(* CODESYS project CintasSoplado.project
   Title: CintasSoplado
   Version: 0.0.0.0
   Author: serbogr1

Project tree, tasks and I/O mapping:
  MyController : TM241CE40R, Schneider Electric, order no. TM241CE40R, version 4.0.6.18
    application Application
      libraries: Toolbox, 2.2.0.0 (Schneider Electric); SysTime, 3.4.1.20 (System)
      task MAST (cyclic, interval 50 ms, priority 15) calls ProcesoUno, ProcesoDos, Pulsadores, PID, ControlSoplado, Gestion_HMI
      global variables GVL
      visualisation HMIW_Control
      image pool ImagePool
      program ProcesoDos [SFC]: E2_active, E10_active
      program PID [LD]
      program ProcesoUno [SFC]: E8_active, E7_active, E9_active, E10_active, E11_active, E12_active, E1_active
      program Pulsadores [LD]
      program ControlSoplado [SFC]: E1_active
      program Gestion_HMI [LD]
    DI : Digital Inputs, Schneider Electric, version 4.0.6.18
        input  idwDI_IDW0 : DWORD  // IDW0
        input  ibDI_IB1 : BYTE  // IB1
    DQ : Digital Outputs, Schneider Electric, version 4.0.6.18
        output qwDQ_QW0 : WORD  // QW0
        output qbDQ_QB1 : BYTE  // QB1
    Counters : Counters, Schneider Electric, version 4.0.6.18
    Pulse_Generators : Pulse Generators, Schneider Electric, version 4.0.6.18
    Cartridge_1 : Cartridge, Schneider Electric, version 4.0.6.18
      TMC4AI2 : TMC4AI2, Schneider Electric, order no. TMC4AI2, version 1.0.1.0
          input  iiTMC4AI2_IW0 : INT  // IW0
          input  iiTMC4AI2_IW1 : INT  // IW1
          input  ibTMC4AI2_IW2 : BYTE  // IW2
    Cartridge_2 : Cartridge, Schneider Electric, version 4.0.6.18
      TMC4AQ2 : TMC4AQ2, Schneider Electric, order no. TMC4AQ2, version 1.0.1.1
          output qiTMC4AQ2_QW0 : INT  // QW0
          output qiTMC4AQ2_QW1 : INT  // QW1
          input  ibTMC4AQ2_IW0 : BYTE  // IW0
    IO_Bus : IO bus - TM3, Schneider Electric, version 4.0.6.18
    COM_Bus : COM bus, Schneider Electric, version 4.0.6.18
    Ethernet_1 : Ethernet Network, Schneider Electric, version 4.0.6.18
        settings: WebServer = TRUE; FTP Server = TRUE; SoMachine Protocol = TRUE; Modbus Server = TRUE; NetManage Protocol = TRUE; SNMP protocol = TRUE; Enable Routing = FALSE; WebVisu protocol = TRUE; DHCP Server Active = FALSE
    Serial_Line_1 : Serial line, Schneider Electric, version 4.0.6.18
      SoMachine_Network_Manager : SoMachine-Network Manager, Schneider Electric, version 4.0.0.2
    Serial_Line_2 : Serial line, Schneider Electric, version 4.0.6.18
      Modbus_Manager : Modbus Manager, Schneider Electric, version 4.0.0.2
  text list GlobalTextList
*)

// MyController/Application/GVL
VAR_GLOBAL
END_VAR

// MyController/Application/ProcesoUno
PROGRAM ProcesoUno
VAR
	bS_FC_Empujador_1          AT %IX0.0: BOOL; (*I1*)
	bS_IC_Empujador_1          AT %IX0.1: BOOL; (*I2*)
	bS_FC_Empujador_2          AT %IX0.2: BOOL; (*I3*)
	bS_IC_Empujador_2          AT %IX0.3: BOOL; (*I4*)
	bS_FT_Empujador_1          AT %IX0.4: BOOL; (*I5*)
	bS_FT_Fresadora            AT %IX0.5: BOOL; (*I6*)
	bS_FT_Carga                AT %IX0.6: BOOL; (*I7*)
	bS_FT_Taladro              AT %IX0.7: BOOL; (*I8*)
	bS_FT_Salida               AT %IX1.0: BOOL; (*I9*)

	FalloSensores              AT %MX0.5: BOOL:=FALSE;;
	CintaFresadoraP1                    : BOOL;	
	CintaTaladroP1                      : BOOL;	
	CintaAlimentacionP1                 : BOOL;
	MotorFresadora                      : BOOL;
    bSiguientePieza            AT %MX0.4: BOOL; (*Activa cuando se puede poner la siguiente pieza*)
	iTiempoFresado                      : INT:=2;	
END_VAR

VAR_OUTPUT
	tEmpujador_1   : TIME:=T#1S;
	tFresado       : TIME:=T#1S;
END_VAR

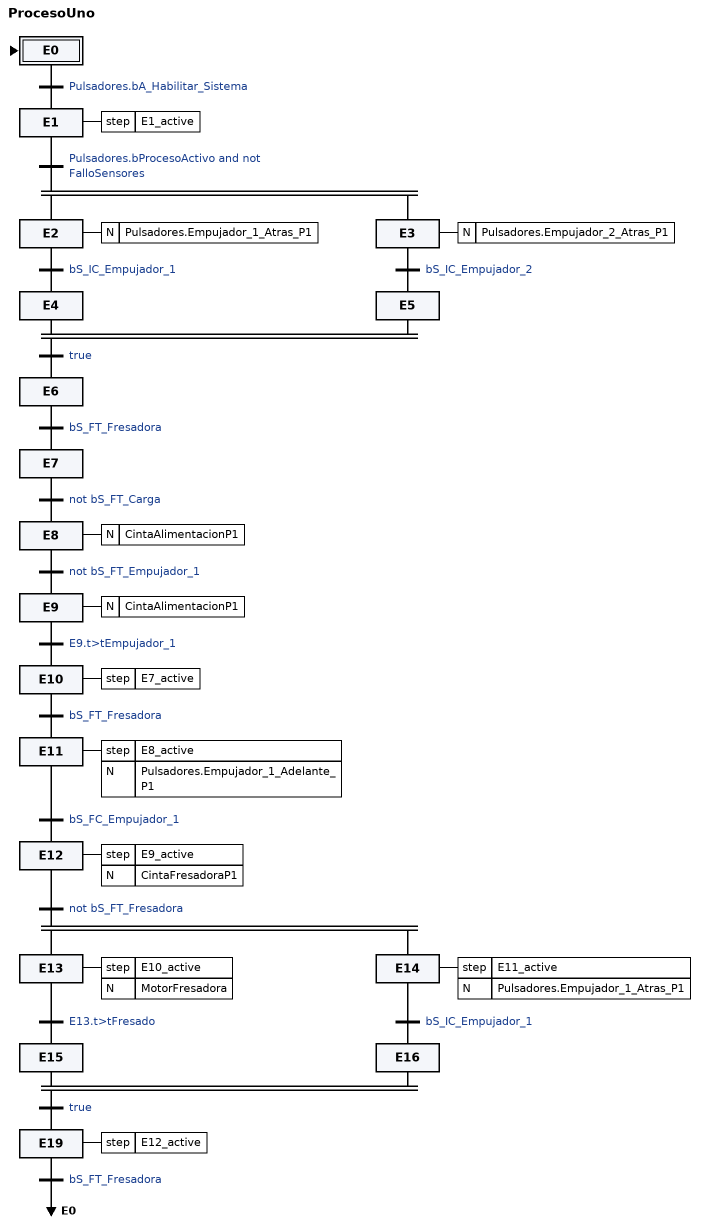
INITIAL_STEP E0:
END_STEP
TRANSITION FROM E0 TO E1
    := Pulsadores.bA_Habilitar_Sistema;
END_TRANSITION
STEP E1:
    E1_active(N);  // step action
END_STEP
TRANSITION FROM E1 TO (E2, E3)
    := Pulsadores.bProcesoActivo and not FalloSensores;
END_TRANSITION
STEP E2:
    Pulsadores.Empujador_1_Atras_P1(N);
END_STEP
TRANSITION FROM E2 TO E4
    := bS_IC_Empujador_1;
END_TRANSITION
STEP E4:
END_STEP
STEP E3:
    Pulsadores.Empujador_2_Atras_P1(N);
END_STEP
TRANSITION FROM E3 TO E5
    := bS_IC_Empujador_2;
END_TRANSITION
STEP E5:
END_STEP
TRANSITION FROM (E4, E5) TO E6
    := true;
END_TRANSITION
STEP E6:
END_STEP
TRANSITION FROM E6 TO E7
    := bS_FT_Fresadora;
END_TRANSITION
STEP E7:
END_STEP
TRANSITION FROM E7 TO E8
    := not bS_FT_Carga;
END_TRANSITION
STEP E8:
    CintaAlimentacionP1(N);
END_STEP
TRANSITION FROM E8 TO E9
    := not bS_FT_Empujador_1;
END_TRANSITION
STEP E9:
    CintaAlimentacionP1(N);
END_STEP
TRANSITION FROM E9 TO E10
    := E9.t>tEmpujador_1;
END_TRANSITION
STEP E10:
    E7_active(N);  // step action
END_STEP
TRANSITION FROM E10 TO E11
    := bS_FT_Fresadora;
END_TRANSITION
STEP E11:
    E8_active(N);  // step action
    Pulsadores.Empujador_1_Adelante_P1(N);
END_STEP
TRANSITION FROM E11 TO E12
    := bS_FC_Empujador_1;
END_TRANSITION
STEP E12:
    E9_active(N);  // step action
    CintaFresadoraP1(N);
END_STEP
TRANSITION FROM E12 TO (E13, E14)
    := not bS_FT_Fresadora;
END_TRANSITION
STEP E13:
    E10_active(N);  // step action
    MotorFresadora(N);
END_STEP
TRANSITION FROM E13 TO E15
    := E13.t>tFresado;
END_TRANSITION
STEP E15:
END_STEP
STEP E14:
    E11_active(N);  // step action
    Pulsadores.Empujador_1_Atras_P1(N);
END_STEP
TRANSITION FROM E14 TO E16
    := bS_IC_Empujador_1;
END_TRANSITION
STEP E16:
END_STEP
TRANSITION FROM (E15, E16) TO E19
    := true;
END_TRANSITION
STEP E19:
    E12_active(N);  // step action
END_STEP
TRANSITION FROM E19 TO E0
    := bS_FT_Fresadora;
END_TRANSITION

ACTION E8_active:
IF bS_FT_Carga THEN
	bSiguientePieza := TRUE;
ELSIF NOT bS_FT_Carga THEN
	bSiguientePieza := FALSE;
END_IF
END_ACTION

ACTION E7_active:
IF bS_FT_Carga THEN
	bSiguientePieza := TRUE;
ELSIF NOT bS_FT_Carga THEN
	bSiguientePieza := FALSE;
END_IF
END_ACTION

ACTION E9_active:
IF bS_FT_Carga THEN
	bSiguientePieza := TRUE;
ELSIF NOT bS_FT_Carga THEN
	bSiguientePieza := FALSE;
END_IF
END_ACTION

ACTION E10_active:
IF bS_FT_Carga THEN
	bSiguientePieza := TRUE;
ELSIF NOT bS_FT_Carga THEN
	bSiguientePieza := FALSE;
END_IF

IF Gestion_HMI.bSum_T_Fresado THEN
	iTiempoFresado := iTiempoFresado + 1;
END_IF
IF Gestion_HMI.bRes_T_Fresado THEN
	iTiempoFresado := iTiempoFresado - 1;
END_IF

	tFresado := INT_TO_TIME(iTiempoFresado*1000);
END_ACTION

ACTION E11_active:
IF bS_FT_Carga THEN
	bSiguientePieza := TRUE;
ELSIF NOT bS_FT_Carga THEN
	bSiguientePieza := FALSE;
END_IF
END_ACTION

ACTION E12_active:
IF bS_FT_Carga THEN
	bSiguientePieza := TRUE;
ELSIF NOT bS_FT_Carga THEN
	bSiguientePieza := FALSE;
END_IF
END_ACTION

ACTION E1_active:
IF NOT Pulsadores.bBotonInicioHMIW THEN
	IF NOT bS_FT_Carga THEN
		FalloSensores:=TRUE;	
	END_IF
	IF NOT bS_FT_Empujador_1 THEN
		FalloSensores:=TRUE;
	END_IF
	IF NOT bS_FT_Fresadora THEN
		FalloSensores:=TRUE;
	END_IF
	IF NOT bS_FT_Taladro THEN
		FalloSensores:=TRUE;
	END_IF
	IF NOT bS_FT_Salida THEN
		FalloSensores:=TRUE;	
	END_IF
	
	IF bS_FT_Carga AND bS_FT_Empujador_1 AND bS_FT_Fresadora AND bS_FT_Taladro AND bS_FT_Salida THEN
		FalloSensores:=FALSE;			
	END_IF
END_IF
END_ACTION

END_PROGRAM

// MyController/Application/Gestion_HMI
PROGRAM Gestion_HMI
VAR
	bSum_T_Fresado              AT %MX3.0: BOOL;
	bRes_T_Fresado              AT %MX3.1: BOOL;
	bSum_T_Taladrado            AT %MX3.2: BOOL;
	bRes_T_Taladrado            AT %MX3.3: BOOL;
	bSum_T_Soplado              AT %MX3.4: BOOL;
	bRes_T_Soplado              AT %MX3.5: BOOL;		
	bSum_AnguloInicio           AT %MX3.6: BOOL;		
	bRes_AnguloInicio           AT %MX3.7: BOOL;
	bSum_AnguloSoplado          AT %MX4.0: BOOL;
	bRes_AnguloSoplado          AT %MX4.1: BOOL;	

	bSe_FC_Empujador_1          AT %MX0.6: BOOL; (*Posición de pieza según el sensor en la HMI*)
	bSe_FC_Empujador_2          AT %MX0.7: BOOL; 
	bSe_FT_Empujador_1          AT %MX1.0: BOOL; 
	bSe_FT_Fresadora            AT %MX1.2: BOOL; 
	bSe_FT_Carga                AT %MX1.3: BOOL; 
	bSe_FT_Taladro              AT %MX1.4: BOOL; 
	bSe_FT_Salida               AT %MX1.5: BOOL; 
	
	bAe_M_Empujador_1_Adelante  AT %MX1.6: BOOL;
	bAe_M_Fresadora             AT %MX1.7: BOOL;
	bAe_M_Taladro               AT %MX2.0: BOOL;
	bAe_M_Empujador_2_Adelante  AT %MX2.1: BOOL;	
	
	iGrados                     AT %MD140: REAL:=ControlSoplado.rActuador/1000;
	rActuadorHMI                AT %MD150: REAL:=ControlSoplado.vActuador;
	rSensorHMI                  AT %MD160: REAL;
END_VAR

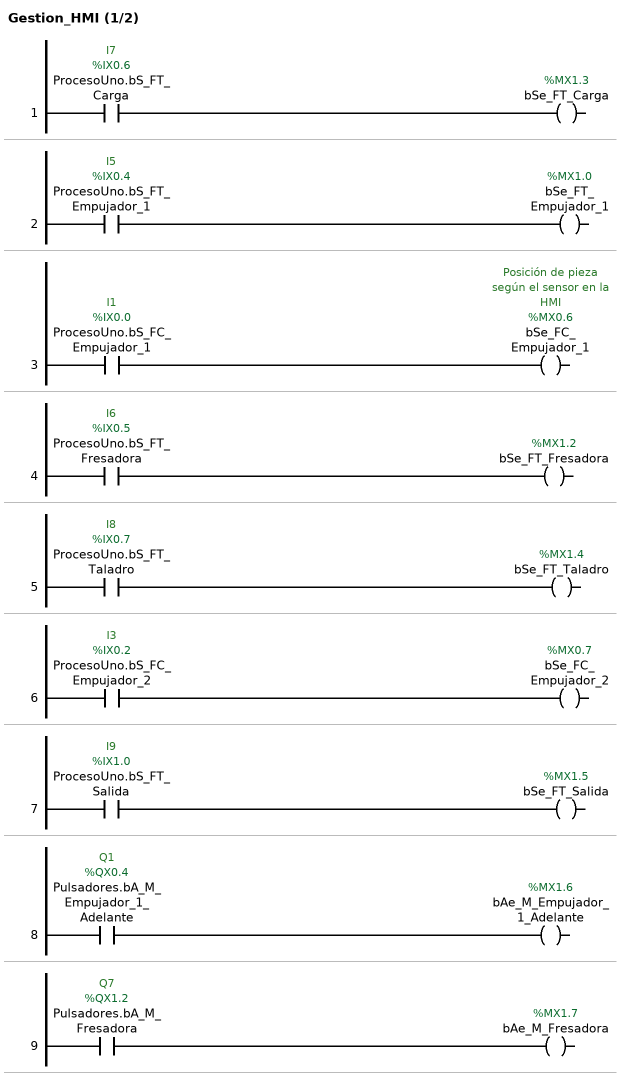
// NETWORK 1
//   ProcesoUno.bS_FT_Carga: I7 | AT %IX0.6
//   bSe_FT_Carga: AT %MX1.3
bSe_FT_Carga := ProcesoUno.bS_FT_Carga;

// NETWORK 2
//   ProcesoUno.bS_FT_Empujador_1: I5 | AT %IX0.4
//   bSe_FT_Empujador_1: AT %MX1.0
bSe_FT_Empujador_1 := ProcesoUno.bS_FT_Empujador_1;

// NETWORK 3
//   ProcesoUno.bS_FC_Empujador_1: I1 | AT %IX0.0
//   bSe_FC_Empujador_1: Posición de pieza según el sensor en la HMI | AT %MX0.6
bSe_FC_Empujador_1 := ProcesoUno.bS_FC_Empujador_1;

// NETWORK 4
//   ProcesoUno.bS_FT_Fresadora: I6 | AT %IX0.5
//   bSe_FT_Fresadora: AT %MX1.2
bSe_FT_Fresadora := ProcesoUno.bS_FT_Fresadora;

// NETWORK 5
//   ProcesoUno.bS_FT_Taladro: I8 | AT %IX0.7
//   bSe_FT_Taladro: AT %MX1.4
bSe_FT_Taladro := ProcesoUno.bS_FT_Taladro;

// NETWORK 6
//   ProcesoUno.bS_FC_Empujador_2: I3 | AT %IX0.2
//   bSe_FC_Empujador_2: AT %MX0.7
bSe_FC_Empujador_2 := ProcesoUno.bS_FC_Empujador_2;

// NETWORK 7
//   ProcesoUno.bS_FT_Salida: I9 | AT %IX1.0
//   bSe_FT_Salida: AT %MX1.5
bSe_FT_Salida := ProcesoUno.bS_FT_Salida;

// NETWORK 8
//   Pulsadores.bA_M_Empujador_1_Adelante: Q1 | AT %QX0.4
//   bAe_M_Empujador_1_Adelante: AT %MX1.6
bAe_M_Empujador_1_Adelante := Pulsadores.bA_M_Empujador_1_Adelante;

// NETWORK 9
//   Pulsadores.bA_M_Fresadora: Q7 | AT %QX1.2
//   bAe_M_Fresadora: AT %MX1.7
bAe_M_Fresadora := Pulsadores.bA_M_Fresadora;

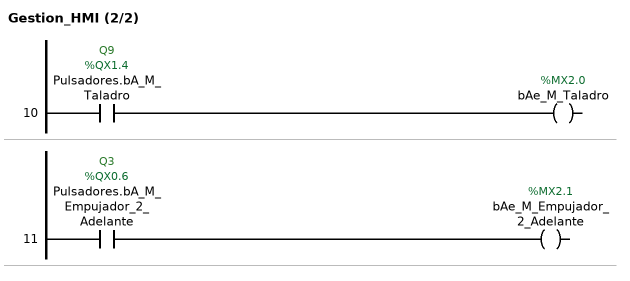
// NETWORK 10
//   Pulsadores.bA_M_Taladro: Q9 | AT %QX1.4
//   bAe_M_Taladro: AT %MX2.0
bAe_M_Taladro := Pulsadores.bA_M_Taladro;

// NETWORK 11
//   Pulsadores.bA_M_Empujador_2_Adelante: Q3 | AT %QX0.6
//   bAe_M_Empujador_2_Adelante: AT %MX2.1
bAe_M_Empujador_2_Adelante := Pulsadores.bA_M_Empujador_2_Adelante;

END_PROGRAM

// MyController/Application/Pulsadores
PROGRAM Pulsadores
VAR
	bA_M_Empujador_1_Adelante  AT %QX0.4: BOOL; (*Q1*)
	bA_M_Empujador_1_Atras     AT %QX0.5: BOOL; (*Q2*)
	bA_M_Empujador_2_Adelante  AT %QX0.6: BOOL; (*Q3*)
	bA_M_Empujador_2_Atras     AT %QX0.7: BOOL; (*Q4*)	
	bA_M_Cinta_Alimentacion    AT %QX1.0: BOOL; (*Q5*)	
	bA_M_Cinta_Fresadora       AT %QX1.1: BOOL; (*Q6*)
	bA_M_Fresadora             AT %QX1.2: BOOL; (*Q7*)	
	bA_M_Cinta_Taladro         AT %QX1.3: BOOL; (*Q8*)	
	bA_M_Taladro               AT %QX1.4: BOOL; (*Q9*)	
	bA_M_Cinta_Salida          AT %QX1.5: BOOL; (*Q10*)		
	bA_Habilitar_Sistema       AT %QX1.6: BOOL; (*Q11*)	
	
	bBotonEmergenciaHMI        AT %MX0.0: BOOL; (*Boton Emergencia HMI*)
	bBotonEmergenciaHMIW                : BOOL; (*Boton Emergencia HMIW*)	
	bBotonEncendidoHMI         AT %MX0.1: BOOL; (*Boton Encendido HMI*)
	bBotonEncendidoHMIW                 : BOOL; (*Boton Encendido HMIW*)		
	bBotonInicioHMI            AT %MX0.2: BOOL; (*Boton Inicio HMI*)
	bBotonInicioHMIW                    : BOOL; (*Boton Inicio HMIW*)	

	bAlarma_ON                 AT %MX0.3: BOOL; (*Activa cuando se pulsa alarma*)
	bProcesoActivo              : BOOL; (*Activa cuando se pulsa inicio*)	
	Empujador_1_Adelante_P1     : BOOL;
	Empujador_1_Adelante_P2     : BOOL;
	Empujador_2_Adelante_P1     : BOOL;	
    Empujador_2_Adelante_P2     : BOOL;
	Empujador_1_Atras_P1        : BOOL;
	Empujador_1_Atras_P2        : BOOL;	
	Empujador_2_Atras_P1        : BOOL;
	Empujador_2_Atras_P2        : BOOL;		
	rLongTime: INT;
END_VAR

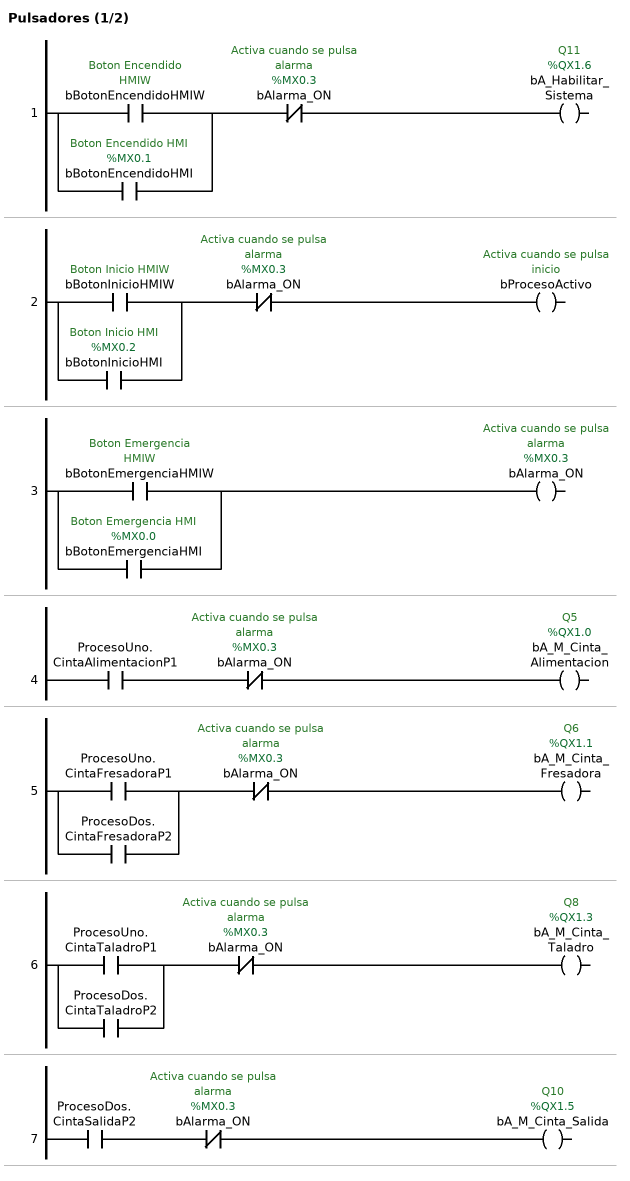
// NETWORK 1
//   bBotonEncendidoHMIW: Boton Encendido HMIW
//   bBotonEncendidoHMI: Boton Encendido HMI | AT %MX0.1
//   bAlarma_ON: Activa cuando se pulsa alarma | AT %MX0.3
//   bA_Habilitar_Sistema: Q11 | AT %QX1.6
bA_Habilitar_Sistema := (bBotonEncendidoHMIW OR bBotonEncendidoHMI) AND NOT bAlarma_ON;

// NETWORK 2
//   bBotonInicioHMIW: Boton Inicio HMIW
//   bBotonInicioHMI: Boton Inicio HMI | AT %MX0.2
//   bAlarma_ON: Activa cuando se pulsa alarma | AT %MX0.3
//   bProcesoActivo: Activa cuando se pulsa inicio
bProcesoActivo := (bBotonInicioHMIW OR bBotonInicioHMI) AND NOT bAlarma_ON;

// NETWORK 3
//   bBotonEmergenciaHMIW: Boton Emergencia HMIW
//   bBotonEmergenciaHMI: Boton Emergencia HMI | AT %MX0.0
//   bAlarma_ON: Activa cuando se pulsa alarma | AT %MX0.3
bAlarma_ON := bBotonEmergenciaHMIW OR bBotonEmergenciaHMI;

// NETWORK 4
//   bAlarma_ON: Activa cuando se pulsa alarma | AT %MX0.3
//   bA_M_Cinta_Alimentacion: Q5 | AT %QX1.0
bA_M_Cinta_Alimentacion := ProcesoUno.CintaAlimentacionP1 AND NOT bAlarma_ON;

// NETWORK 5
//   bAlarma_ON: Activa cuando se pulsa alarma | AT %MX0.3
//   bA_M_Cinta_Fresadora: Q6 | AT %QX1.1
bA_M_Cinta_Fresadora := (ProcesoUno.CintaFresadoraP1 OR ProcesoDos.CintaFresadoraP2) AND NOT bAlarma_ON;

// NETWORK 6
//   bAlarma_ON: Activa cuando se pulsa alarma | AT %MX0.3
//   bA_M_Cinta_Taladro: Q8 | AT %QX1.3
bA_M_Cinta_Taladro := (ProcesoUno.CintaTaladroP1 OR ProcesoDos.CintaTaladroP2) AND NOT bAlarma_ON;

// NETWORK 7
//   bAlarma_ON: Activa cuando se pulsa alarma | AT %MX0.3
//   bA_M_Cinta_Salida: Q10 | AT %QX1.5
bA_M_Cinta_Salida := ProcesoDos.CintaSalidaP2 AND NOT bAlarma_ON;

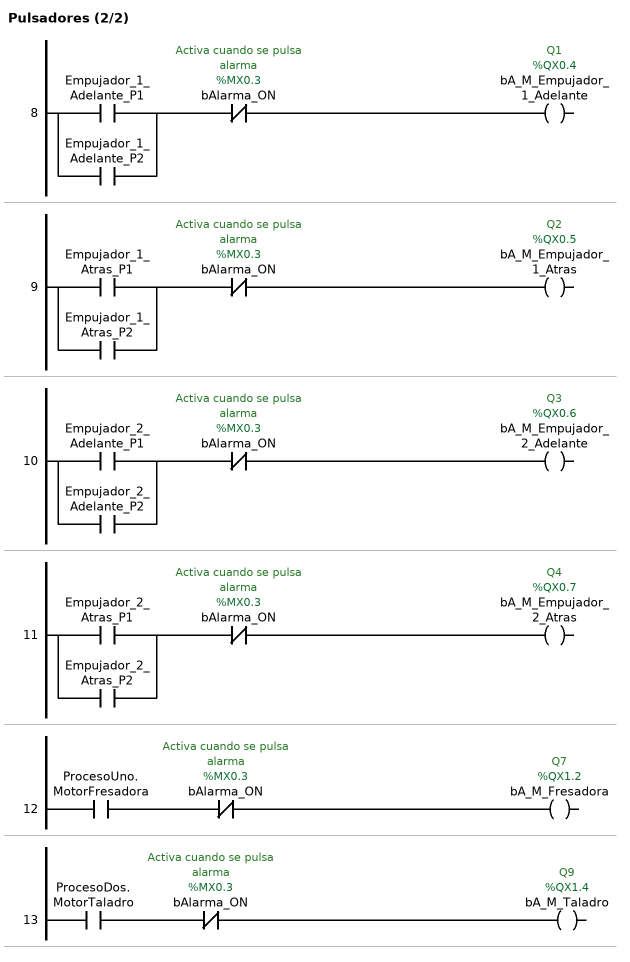
// NETWORK 8
//   bAlarma_ON: Activa cuando se pulsa alarma | AT %MX0.3
//   bA_M_Empujador_1_Adelante: Q1 | AT %QX0.4
bA_M_Empujador_1_Adelante := (Empujador_1_Adelante_P1 OR Empujador_1_Adelante_P2) AND NOT bAlarma_ON;

// NETWORK 9
//   bAlarma_ON: Activa cuando se pulsa alarma | AT %MX0.3
//   bA_M_Empujador_1_Atras: Q2 | AT %QX0.5
bA_M_Empujador_1_Atras := (Empujador_1_Atras_P1 OR Empujador_1_Atras_P2) AND NOT bAlarma_ON;

// NETWORK 10
//   bAlarma_ON: Activa cuando se pulsa alarma | AT %MX0.3
//   bA_M_Empujador_2_Adelante: Q3 | AT %QX0.6
bA_M_Empujador_2_Adelante := (Empujador_2_Adelante_P1 OR Empujador_2_Adelante_P2) AND NOT bAlarma_ON;

// NETWORK 11
//   bAlarma_ON: Activa cuando se pulsa alarma | AT %MX0.3
//   bA_M_Empujador_2_Atras: Q4 | AT %QX0.7
bA_M_Empujador_2_Atras := (Empujador_2_Atras_P1 OR Empujador_2_Atras_P2) AND NOT bAlarma_ON;

// NETWORK 12
//   bAlarma_ON: Activa cuando se pulsa alarma | AT %MX0.3
//   bA_M_Fresadora: Q7 | AT %QX1.2
bA_M_Fresadora := ProcesoUno.MotorFresadora AND NOT bAlarma_ON;

// NETWORK 13
//   bAlarma_ON: Activa cuando se pulsa alarma | AT %MX0.3
//   bA_M_Taladro: Q9 | AT %QX1.4
bA_M_Taladro := ProcesoDos.MotorTaladro AND NOT bAlarma_ON;

END_PROGRAM

// MyController/Application/ProcesoDos
PROGRAM ProcesoDos
VAR
    CintaSalidaP2                : BOOL;
    MotorTaladro                 : BOOL;
	CintaFresadoraP2             : BOOL;
	CintaTaladroP2               : BOOL;	
	iTiempoTaladrado    AT %MW110: INT:=2;
	rPiezasTerminadas            : INT:=0;		
	tTaladrado                   : TIME:=T#2S;
	tEmpujador_2                 : TIME:=T#2S;	
END_VAR

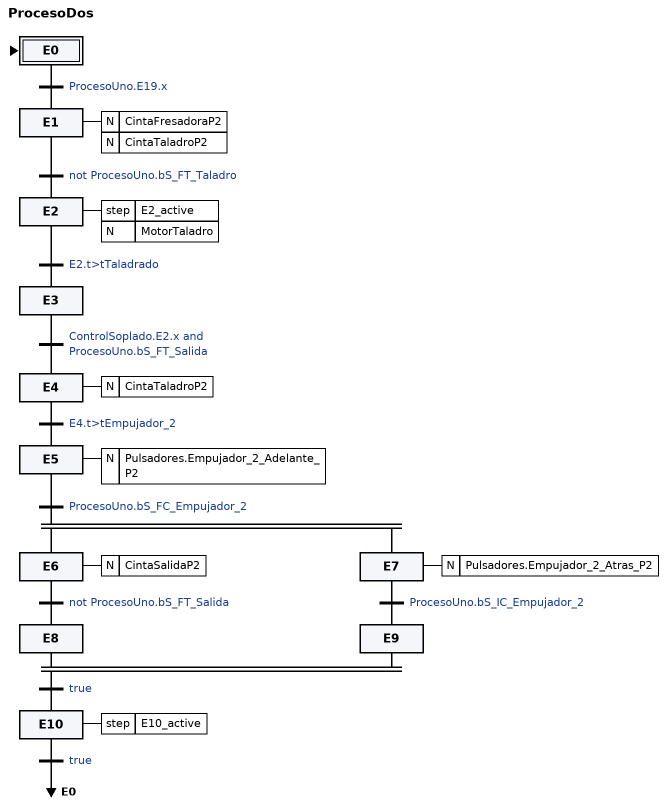
INITIAL_STEP E0:
END_STEP
TRANSITION FROM E0 TO E1
    := ProcesoUno.E19.x;
END_TRANSITION
STEP E1:
    CintaFresadoraP2(N);
    CintaTaladroP2(N);
END_STEP
TRANSITION FROM E1 TO E2
    := not ProcesoUno.bS_FT_Taladro;
END_TRANSITION
STEP E2:
    E2_active(N);  // step action
    MotorTaladro(N);
END_STEP
TRANSITION FROM E2 TO E3
    := E2.t>tTaladrado;
END_TRANSITION
STEP E3:
END_STEP
TRANSITION FROM E3 TO E4
    := ControlSoplado.E2.x and ProcesoUno.bS_FT_Salida;
END_TRANSITION
STEP E4:
    CintaTaladroP2(N);
END_STEP
TRANSITION FROM E4 TO E5
    := E4.t>tEmpujador_2;
END_TRANSITION
STEP E5:
    Pulsadores.Empujador_2_Adelante_P2(N);
END_STEP
TRANSITION FROM E5 TO (E6, E7)
    := ProcesoUno.bS_FC_Empujador_2;
END_TRANSITION
STEP E6:
    CintaSalidaP2(N);
END_STEP
TRANSITION FROM E6 TO E8
    := not ProcesoUno.bS_FT_Salida;
END_TRANSITION
STEP E8:
END_STEP
STEP E7:
    Pulsadores.Empujador_2_Atras_P2(N);
END_STEP
TRANSITION FROM E7 TO E9
    := ProcesoUno.bS_IC_Empujador_2;
END_TRANSITION
STEP E9:
END_STEP
TRANSITION FROM (E8, E9) TO E10
    := true;
END_TRANSITION
STEP E10:
    E10_active(N);  // step action
END_STEP
TRANSITION FROM E10 TO E0
    := true;
END_TRANSITION

ACTION E2_active:
  
IF Gestion_HMI.bSum_T_Taladrado THEN
	iTiempoTaladrado := iTiempoTaladrado + 1;
END_IF
IF Gestion_HMI.bRes_T_Taladrado THEN
	iTiempoTaladrado := iTiempoTaladrado - 1;
END_IF

	tTaladrado := INT_TO_TIME(iTiempoTaladrado*1000);
END_ACTION

ACTION E10_active:
IF NOT ProcesoUno.bS_FT_Salida THEN
	rPiezasTerminadas := rPiezasTerminadas + 1;
END_IF
END_ACTION

END_PROGRAM

// MyController/Application/ControlSoplado
PROGRAM ControlSoplado
VAR
	bCS_FinSoplado                 : BOOL:= FALSE;
	vActuador              AT %QW4 : WORD;	
	rActuador                      : REAL:=0;
	iPosReposo                     : INT:=0;
	iPosInicio                     : REAL:=3300;
	iPosSoplado                    : REAL:=5000;	
	iPosInicioGrados               : REAL:=25;
	iPosSopladoGrados              : REAL:=45;		
    step                           : INT:=1;
	next_step                      : INT:=1;
	iTiempoSoplado        AT %MW120: INT:=2;	
	tTiempoSoplado                 : TIME:=T#2S;	
	TimeSET                      : INT:=0;

	MyTimer: INT;
	StartTimer: INT;
	MyMSeconds: DINT;
	
	MY_TON: TON;
	IN_VALUE: BOOL:=false;
	TIME_SET: TIME:=t#5000ms;
END_VAR

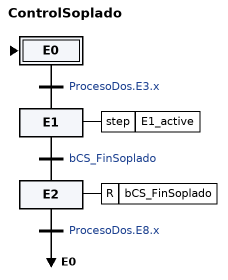
INITIAL_STEP E0:
END_STEP
TRANSITION FROM E0 TO E1
    := ProcesoDos.E3.x;
END_TRANSITION
STEP E1:
    E1_active(N);  // step action
END_STEP
TRANSITION FROM E1 TO E2
    := bCS_FinSoplado;
END_TRANSITION
STEP E2:
    bCS_FinSoplado(R);
END_STEP
TRANSITION FROM E2 TO E0
    := ProcesoDos.E8.x;
END_TRANSITION

ACTION E1_active:

MY_TON(IN:= IN_VALUE,PT:= TIME_SET);
(*IN_VALUE - is BOOL variable that activates your timer
  TIME_SET - is TIME variable*)

IF Gestion_HMI.bSum_T_Soplado THEN              (*Incremento/dexcremento desde HMI el tiempo de soplado*)
	iTiempoSoplado := iTiempoSoplado + 1;
END_IF
IF Gestion_HMI.bRes_T_Soplado THEN
	iTiempoSoplado := iTiempoSoplado - 1;
END_IF

IF Gestion_HMI.bSum_AnguloInicio THEN           (*Incremento/dexcremento desde HMI el angulo de inicio*)
	iPosInicioGrados := iPosInicioGrados + 1;
END_IF
IF Gestion_HMI.bRes_AnguloInicio THEN
	iPosInicioGrados := iPosInicioGrados - 1;
END_IF

IF Gestion_HMI.bSum_AnguloSoplado THEN           (*Incremento/dexcremento desde HMI el angulo de soplado*)
	iPosSopladoGrados := iPosSopladoGrados + 1;
END_IF
IF Gestion_HMI.bRes_AnguloSoplado THEN
	iPosSopladoGrados := iPosSopladoGrados - 1;
END_IF

tTiempoSoplado := INT_TO_TIME(iTiempoSoplado*1000);

iPosInicio :=  109.09 * iPosInicioGrados;         (*Conversión de grados del spinControl a tensión x 1000*)
iPosSoplado := 109.09 * iPosSopladoGrados;

IF ControlSoplado.E1.x THEN
	CASE step OF
		1:                                            (*Llevar hélice a posición de inicio*)
			WHILE vActuador < iPosInicio DO
				rActuador := rActuador + 100;
				vActuador := REAL_TO_WORD(rActuador);



	
WHILE TimeSET < 4 DO
	IN_VALUE:=TRUE;
	IF MY_TON.Q THEN
		TimeSET := TimeSET +1;
		IN_VALUE:=FALSE;		
	END_IF	
END_WHILE

		
			END_WHILE

			step:=2;
	    2:                                           (*Llevar hélice a posición de soplado*)
			WHILE vActuador < iPosSoplado DO
				rActuador := rActuador + 100;
				vActuador := REAL_TO_WORD(rActuador);

			END_WHILE

			step:=3;
		3:                                           (*Llevar hélice a posición de reposo*)
			WHILE vActuador > iPosReposo DO
				rActuador := rActuador - 100;
				vActuador := REAL_TO_WORD(rActuador);

			END_WHILE
			step:=4;
		4:                                           (*Señal de fin de soplado*)
			bCS_FinSoplado:=TRUE;
			step:=1;
		ELSE
			bCS_FinSoplado:=FALSE;
			step:=1;
	END_CASE	
END_IF
END_ACTION

END_PROGRAM

// MyController/Application/PID
PROGRAM PID
VAR
	vActuador_PID            : WORD;
	rActuador                : REAL;
	vSensor          AT %IW3 : WORD;	
	rSensor                  : REAL;	
	rReferencia              : REAL:=-26;
	AutoManual               : BOOL;
	ResetPID                 : BOOL;
	FB_Scaling_vS            : FB_Scaling; (*Escalado para tensión del sensor*)
	FB_Scaling_vA            : FB_Scaling; (*Escalado para tensión al actuador*)
	PID_ControHelice         : Util.PID;
END_VAR

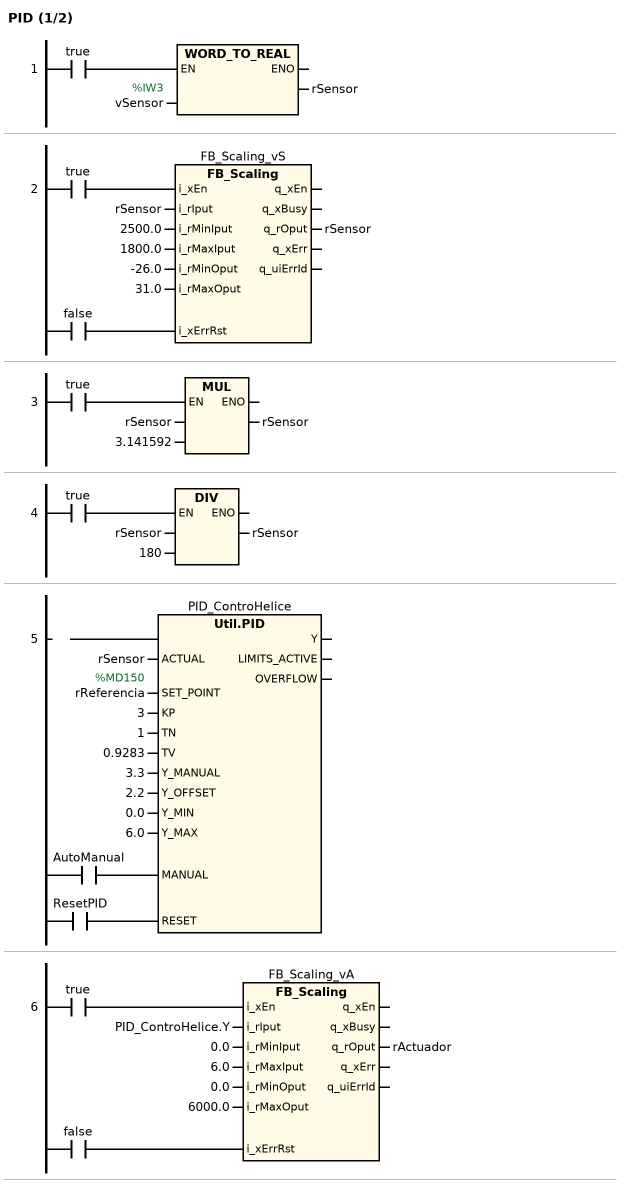
// NETWORK 1
//   vSensor: AT %IW3
IF true THEN rSensor := WORD_TO_REAL(vSensor); END_IF

// NETWORK 2
//   FB_Scaling_vS: Escalado para tensión del sensor
FB_Scaling_vS(
    i_xEn := true,
    i_rIput := rSensor,
    i_rMinIput := 2500.0,
    i_rMaxIput := 1800.0,
    i_rMinOput := -26.0,
    i_rMaxOput := 31.0,
    i_xErrRst := false,
    q_rOput => rSensor); // FB_Scaling

// NETWORK 3
IF true THEN rSensor := rSensor * 3.141592; END_IF

// NETWORK 4
IF true THEN rSensor := rSensor / 180; END_IF

// NETWORK 5
//   rReferencia: AT %MD150
PID_ControHelice(
    ACTUAL := rSensor,
    SET_POINT := rReferencia,
    KP := 3,
    TN := 1,
    TV := 0.9283,
    Y_MANUAL := 3.3,
    Y_OFFSET := 2.2,
    Y_MIN := 0.0,
    Y_MAX := 6.0,
    MANUAL := AutoManual,
    RESET := ResetPID); // Util.PID

// NETWORK 6
//   FB_Scaling_vA: Escalado para tensión al actuador
//   PID_ControHelice.Y: manipulated variable, set value
FB_Scaling_vA(
    i_xEn := true,
    i_rIput := PID_ControHelice.Y,
    i_rMinIput := 0.0,
    i_rMaxIput := 6.0,
    i_rMinOput := 0.0,
    i_rMaxOput := 6000.0,
    i_xErrRst := false,
    q_rOput => rActuador); // FB_Scaling

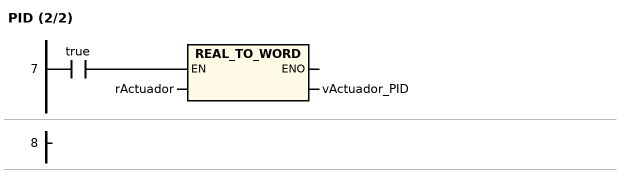
// NETWORK 7
IF true THEN vActuador_PID := REAL_TO_WORD(rActuador); END_IF

// NETWORK 8

END_PROGRAM

// MyController/Application/HMIW_Control
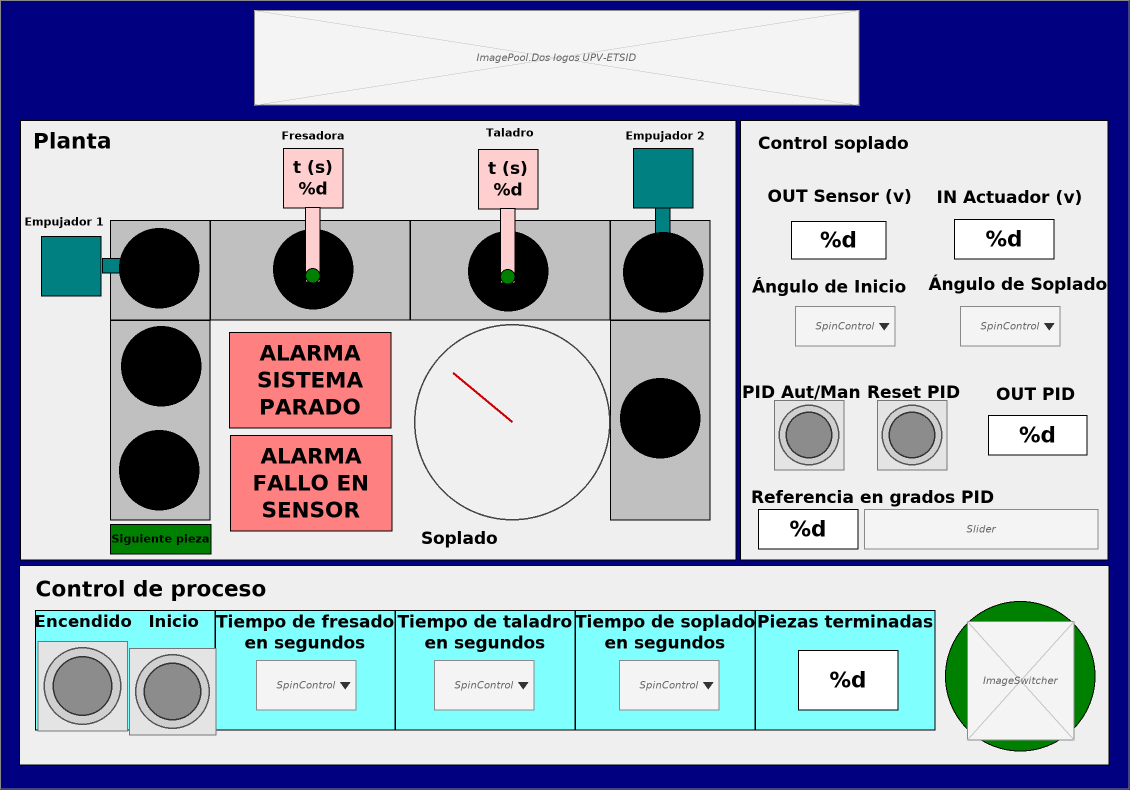
VISUALIZATION HMIW_Control  // 1130x790
    Rectangle (740,120 368x440)
    Rectangle (20,120 716x440)
    Rectangle (19,565 1090x200)
    Rectangle (110,220 100x100)
    Rectangle (110,320 100x200)
    Rectangle (610,320 100x200)
    Rectangle (610,220 100x100)
    Rectangle (210,220 200x100)
    Rectangle (410,220 200x100)
    Rectangle (35,610 180x120), "Encendido Inicio"
    Rectangle (215,610 180x120), "Tiempo de fresado en segundos"
    Rectangle (395,610 180x120), "Tiempo de taladro en segundos"
    Rectangle (575,610 180x120), "Tiempo de soplado en segundos"
    Rectangle (755,610 180x120), "Piezas terminadas"
    Label (40,574 222x30), "Control de proceso"
    SpinControl (256,660 100x50), variable: ProcesoUno.iTiempoFresado
    SpinControl (434,660 100x50), variable: ProcesoDos.iTiempoTaladrado
    SpinControl (619,660 100x50), variable: ControlSoplado.iTiempoSoplado
    PushSwitchLed (37,641 91x90), variable: Pulsadores.bBotonEncendidoHMIW, behaviour: TOGGLE, style: Switch-PushSwitchLed-Gray
    Ellipse (119,430 80x80), invisible if: ProcesoUno.bS_FT_Carga
    Ellipse (121,326 80x80), invisible if: ProcesoUno.bS_FT_Empujador_1
    Ellipse (273,229 80x80), invisible if: ProcesoUno.bS_FT_Fresadora
    Ellipse (468,231 80x80), invisible if: ProcesoUno.bS_FT_Taladro
    Ellipse (620,378 80x80), invisible if: ProcesoUno.bS_FT_Salida
    RoundedRectangle (798,650 100x60), "%d", text variable: ProcesoDos.rPiezasTerminadas
    RoundedRectangle (41,236 60x60)
    RoundedRectangle (283,148 60x60), "t (s) %d", text variable: ProcesoUno.E13.t/1000, colour toggle: ProcesoUno.MotorFresadora
    RoundedRectangle (478,149 60x60), "t (s) %d", text variable: ProcesoDos.E2.t/1000, colour toggle: ProcesoDos.MotorTaladro
    Rectangle (305,207 15x75), colour toggle: ProcesoUno.MotorFresadora
    Rectangle (500,208 15x75), colour toggle: ProcesoDos.MotorTaladro
    Rectangle (655,205 15x75), invisible if: not Pulsadores.bA_M_Empujador_2_Adelante
    Ellipse (305,268 15x15), colour toggle: ProcesoUno.MotorFresadora
    Ellipse (500,269 15x15), colour toggle: ProcesoDos.MotorTaladro
    Rectangle (102,258 75x15), invisible if: not Pulsadores.bA_M_Empujador_1_Adelante
    Ellipse (623,232 80x80), invisible if: ProcesoUno.bS_IC_Empujador_2
    Label (277,121 72x30), "Fresadora"
    Label (23,207 82x30), "Empujador 1"
    Label (475,118 70x30), "Taladro"
    Label (629,121 72x30), "Empujador 2"
    Image (254,10 605x95), image: ImagePool.Dos logos UPV-ETSID
    Label (27,127 91x28), "Planta"
    Ellipse (945,601 150x150), colour toggle: Pulsadores.bBotonEmergenciaHMIW
    ImageSwitcher (967,621 107x119), variable: Pulsadores.bBotonEmergenciaHMIW, background image: ImagePool.BotonEmergencia, image: ImagePool.BotonEmergencia, behaviour: TOGGLE
    RoundedRectangle (110,524 101x30), "Siguiente pieza", colour toggle: ProcesoUno.bSiguientePieza
    Label (766,181 148x30), "OUT Sensor (v)"
    Label (751,482 243x30), "Referencia en grados PID"
    Label (936,182 147x30), "IN Actuador (v)"
    Label (972,379 127x30), "OUT PID"
    RoundedRectangle (791,221 95x38), "%d", text variable: PID.vSensor
    RoundedRectangle (954,219 100x40), "%d", text variable: ControlSoplado.vActuador
    RoundedRectangle (758,509 100x40), "%d", text variable: PID.rReferencia
    Label (751,128 165x30), "Control soplado"
    PushSwitchLed (129,641 87x101), variable: Pulsadores.bBotonInicioHMIW, behaviour: TOGGLE, style: Switch-PushSwitchLed-Gray
    Meter90 (413,324 198x196), value: ControlSoplado.rActuador/1000, style: Meter-Meter90-Gray, scale format: %d, scale 0..60
    Slider (864,509 234x40), variable: PID.rReferencia, scale -26..31
    RoundedRectangle (988,415 99x40), "%d", text variable: PID.vActuador_PID
    SpinControl (795,306 100x40), variable: ControlSoplado.iPosInicioGrados
    SpinControl (960,306 100x40), variable: ControlSoplado.iPosSopladoGrados
    Label (756,272 152x29), "Ángulo de Inicio"
    Label (928,269 180x30), "Ángulo de Soplado"
    RoundedRectangle (229,332 162x96), "ALARMA SISTEMA PARADO", invisible if: not Pulsadores.bAlarma_ON
    RoundedRectangle (230,435 162x96), "ALARMA FALLO EN SENSOR", invisible if: not ProcesoUno.FalloSensores
    Ellipse (119,228 80x80), invisible if: ProcesoUno.bS_IC_Empujador_1
    PushSwitch (877,400 70x70), variable: PID.ResetPID, behaviour: TAP, style: Switch-PushSwitch-Gray
    Label (850,377 127x30), "Reset PID"
    Label (738,377 127x30), "PID Aut/Man"
    PushSwitchLed (774,400 70x70), variable: PID.AutoManual, behaviour: TOGGLE, style: Switch-PushSwitchLed-Gray
    Label (385,523 149x30), "Soplado"
    RoundedRectangle (633,148 60x60)
END_VISUALIZATION
